ORGANIZATION_BLOCK "OB_TEST_AUTO"
TITLE = "Test Main — Simulacion Automatica TGBT V1.0"
{ S7_Optimized_Access := 'TRUE' }
// ============================================================================
// OB_TEST_AUTO  Ver 1.0  2026-03-13
//
// PROPÓSITO:
//   Validar la secuencia automática RED ↔ GD sin hardware real.
//   Reemplaza a OB1 (Main) durante la fase de prueba en taller/laboratorio.
//
// CÓMO ACTIVARLO EN TIA PORTAL (S7-1200):
//   1. Crear este bloque como "Organization Block → Program cycle" con un
//      número diferente a OB1 (ej: OB123).
//   2. En las propiedades de OB1 (Main), marcar "Unlinked" o agregar una
//      condición de retorno inmediato al inicio del bloque (IF NOT TEST_MODE THEN RETURN)
//      para que sólo corra uno de los dos ciclos.
//   3. Alternativamente: renombrar el "Main" actual y asignar este bloque
//      como el nuevo ciclo principal (número de OB = 1).
//
//   IMPORTANTE: NO ejecutar ambos OBs simultáneamente — ambos escriben
//   sobre las mismas instancias (02_FB_SCMTA_DB, 04_FB_CMD_ARBITER_DB, etc.)
//   lo que generaría resultados imprevisibles.
//
// QUÉ HACE ESTE OB vs OB1 (Main):
//   ✓ Llama a TEST_AUTO_FB en lugar de IO_NORMALIZE + Modbus Manager.
//     TEST_AUTO_FB inyecta directamente en DATA_BUFF:
//       - Mediciones de red simuladas (380V/50Hz ↔ 0V/0Hz)
//       - Señales GD1/GD2 (READY/RUNNING) como respuesta a %Q1.0/%Q1.1
//       - Feedback de interruptores como respuesta a pulsos %Q0.x
//   ✓ Llama a SCMTA con timers acortados:
//       T_MIN_GD_STAY  = 60 s   (producción: 10 min)
//       T_GRID_STABLE  = 30 s   (producción: 120 s)
//       T_GD_COOLDOWN  = 10 s   (producción: 60 s)
//   ✓ Llama a SHED, CMD_ARBITER, PULSE_EXPANDER, OUTPUTS igual que OB1.
//   ✗ NO llama a Modbus Manager (sin PM5350P).
//   ✗ NO llama a IO_NORMALIZE (TEST_AUTO_FB reemplaza esa función).
//
// CICLO DE PRUEBA AUTOMÁTICO (configurable en TEST_AUTO_DB):
//   T_FASE_GRID_OK  (30s) → RED OK  → SCMTA = ST_NORMAL_ON_GRID
//   Fin del timer          → RED FALLA (0V) → SCMTA inicia transferencia a GD
//   T_BRK_CONFIRM  (0.6s) → QT1 confirma apertura
//   Abre Q22               → T_BRK_CONFIRM → Q22 confirma apertura
//   T_START_GD_DELAY(3s)   → Arranque GD1 (%Q1.0←TRUE)
//   T_GD1_STARTUP  (8s)   → GD1_READY=TRUE, GD1_RUNNING=TRUE
//   T_GD_STABILIZATION(5s)→ SCMTA cierra QG1
//   T_BRK_CONFIRM  (0.6s) → QG1 confirma cierre → ST_ON_GD1
//   T_MIN_GD_STAY (60s)   → Espera mínima en GD antes de retorno
//   T_FASE_GRID_FAIL(90s) → Red se restaura (380V/50Hz)
//   T_GRID_STABLE  (30s)  → SCMTA abre QG1, cierra Q22, cierra QT1 → ST_ON_GRID
//   Ciclo se repite.
//
// CONTROLES HMI DURANTE PRUEBA (escribir en TEST_AUTO_DB):
//   TEST_AUTO_DB.FORCE_GRID_FAIL  := TRUE  → falla de red inmediata
//   TEST_AUTO_DB.FORCE_GRID_OK    := TRUE  → red restaurada inmediata
//   TEST_AUTO_DB.FORCE_GD1_ALARM  := TRUE  → alarma GD1 en marcha
//   DATA_BUFF.RESET_FAULT         := TRUE  → reset falla SCMTA
// ============================================================================
VERSION : 0.1

BEGIN

    // ========================================================================
    // NETWORK 1: IO REAL (CPU + EXPANSION)
    // Igual que OB1, pero forzando MODE_AUTO para prueba automática.
    // ========================================================================
    "01_FB_IO_NORMALIZE_DB"(
        DI_SYS_AUTO       := TRUE,

        // QT1 (CPU)
        DI_QT1_REMOTE     := %I0.0,
        DI_QT1_CLOSE      := %I0.1,
        DI_QT1_FAULT      := %I0.2,
        DI_QT1_UV_OV      := %I0.3,

        DI_BUSBAR_UV_OV   := %I0.4,

        // QG1 (CPU)
        DI_QG1_REMOTE     := %I0.5,
        DI_QG1_CLOSE      := %I0.6,
        DI_QG1_FAULT      := %I0.7,
        DI_QG1_UV_OV      := %I1.0,

        // QG2 (CPU)
        DI_QG2_REMOTE     := %I1.1,
        DI_QG2_CLOSE      := %I1.2,
        DI_QG2_FAULT      := %I1.3,
        DI_QG2_UV_OV      := %I1.4,

        // Q22 remoto (CPU)
        DI_Q22_REMOTE     := %I1.5,

        MODE_AUTO         => "DATA_BUFF".MODE_AUTO,
        MODE_MANUAL       => "DATA_BUFF".MODE_MANUAL,
        DIAG_MODE_VALID   => "DATA_BUFF".DIAG_MODE_VALID,

        QT1_CLOSED        => "DATA_BUFF".QT1_CLOSED,
        QT1_OPEN          => "DATA_BUFF".QT1_OPEN,
        QT1_FAULT         => "DATA_BUFF".QT1_FAULT,
        QT1_REMOTE        => "DATA_BUFF".QT1_REMOTE,
        QT1_UV_OV_DI      => "DATA_BUFF".QT1_UV_OV_DI,

        BUSBAR_UV_OV_DI   => "DATA_BUFF".BUSBAR_UV_OV_DI,

        QG1_CLOSED        => "DATA_BUFF".QG1_CLOSED,
        QG1_OPEN          => "DATA_BUFF".QG1_OPEN,
        QG1_FAULT         => "DATA_BUFF".QG1_FAULT,
        QG1_REMOTE        => "DATA_BUFF".QG1_REMOTE,
        QG1_UV_OV_DI      => "DATA_BUFF".QG1_UV_OV_DI,

        QG2_CLOSED        => "DATA_BUFF".QG2_CLOSED,
        QG2_OPEN          => "DATA_BUFF".QG2_OPEN,
        QG2_FAULT         => "DATA_BUFF".QG2_FAULT,
        QG2_REMOTE        => "DATA_BUFF".QG2_REMOTE,
        QG2_UV_OV_DI      => "DATA_BUFF".QG2_UV_OV_DI,

        Q22_REMOTE        => "DATA_BUFF".Q22_REMOTE
    );

    // En prueba usar la condición REMOTO real de DI, sin forzado.
    "DATA_BUFF".QT1_REMOTE_ALLOWED := "DATA_BUFF".QT1_REMOTE;
    "DATA_BUFF".QG1_REMOTE_ALLOWED := "DATA_BUFF".QG1_REMOTE;
    "DATA_BUFF".QG2_REMOTE_ALLOWED := "DATA_BUFF".QG2_REMOTE;
    "DATA_BUFF".Q22_REMOTE_ALLOWED := "DATA_BUFF".Q22_REMOTE;
    "DATA_BUFF".Q22_CLOSED := %I8.0;
    "DATA_BUFF".Q22_FAULT  := %I8.1;


    // ========================================================================
    // NETWORK 2: SIMULADOR DE RED/GD
    // Mantiene test automático de transferencia sin depender de Modbus real.
    // ========================================================================
    // Usar parámetros guardados en TEST_AUTO_DB para permitir ajuste online
    // (FORCE_GRID_FAIL, FORCE_GRID_OK, FORCE_GDx_ALARM, tiempos, etc.).
    "TEST_AUTO_DB"();


    // ========================================================================
    // NETWORK 3: MÁQUINA DE ESTADOS SCMTA
    // Misma instancia que OB1 → misma lógica de transferencia.
    // Timers reducidos para hacer el ciclo de prueba razonablemente rápido.
    // ========================================================================
    "02_FB_SCMTA_DB"(
        ENABLE               := TRUE,
        MODE_AUTO            := "DATA_BUFF".MODE_AUTO,
        ENABLE_QG2           := "DB_PARAMS".ENABLE_QG2,
        ENABLE_AUTO_RETURN   := TRUE,
        RESET_FAULT          := "DATA_BUFF".RESET_FAULT,

        // Posición/estado interruptores (provistos por TEST_AUTO_FB)
        QT1_CLOSED           := "DATA_BUFF".QT1_CLOSED,
        QT1_FAULT            := "DATA_BUFF".QT1_FAULT,
        QT1_REMOTE           := "DATA_BUFF".QT1_REMOTE,
        QT1_UV_OV_DI         := "DATA_BUFF".QT1_UV_OV_DI,

        QG1_CLOSED           := "DATA_BUFF".QG1_CLOSED,
        QG1_FAULT            := "DATA_BUFF".QG1_FAULT,
        QG1_REMOTE           := "DATA_BUFF".QG1_REMOTE,

        QG2_CLOSED           := "DATA_BUFF".QG2_CLOSED,
        QG2_FAULT            := "DATA_BUFF".QG2_FAULT,
        QG2_REMOTE           := "DATA_BUFF".QG2_REMOTE,

        Q22_CLOSED           := "DATA_BUFF".Q22_CLOSED,

        // Mediciones RED (provistos por TEST_AUTO_FB — sin Modbus)
        GRID_V_L1L2          := "DATA_BUFF".GRID_V_L1L2,
        GRID_V_L2L3          := "DATA_BUFF".GRID_V_L2L3,
        GRID_V_L3L1          := "DATA_BUFF".GRID_V_L3L1,
        GRID_FREQ            := "DATA_BUFF".GRID_FREQ,
        GRID_MEASUREMENT_OK  := "DATA_BUFF".GRID_MEASUREMENT_OK,
        GRID_PHASE_LOSS      := "DATA_BUFF".GRID_PHASE_LOSS,
        GRID_ALM_UV          := "DATA_BUFF".GRID_ALM_UV,
        GRID_ALM_OV          := "DATA_BUFF".GRID_ALM_OV,

        // Criterio GD por medicion electrica + Modbus OK (simulado por TEST_AUTO_FB)
        GD1_V_L1L2           := "DATA_BUFF".GD1_V_L1L2,
        GD1_V_L2L3           := "DATA_BUFF".GD1_V_L2L3,
        GD1_V_L3L1           := "DATA_BUFF".GD1_V_L3L1,
        GD1_FREQ             := "DATA_BUFF".GD1_FREQ,
        GD1_MEASUREMENT_OK   := "DATA_BUFF".GD1_MEASUREMENT_OK,
        GD2_V_L1L2           := "DATA_BUFF".GD2_V_L1L2,
        GD2_V_L2L3           := "DATA_BUFF".GD2_V_L2L3,
        GD2_V_L3L1           := "DATA_BUFF".GD2_V_L3L1,
        GD2_FREQ             := "DATA_BUFF".GD2_FREQ,
        GD2_MEASUREMENT_OK   := "DATA_BUFF".GD2_MEASUREMENT_OK,

        // Parámetros nominales de red (valores reales)
        V_NOM                := 380.0,
        V_MIN_PCT            := 85.0,
        V_MAX_PCT            := 110.0,
        FREQ_NOM             := 50.0,
        FREQ_MIN             := 49.0,
        FREQ_MAX             := 51.0,

        // Timers de transferencia RED→GD (valores reales de producción)
        T_OPEN_QT1           := T#3s,
        T_OPEN_Q22           := T#3s,
        T_DELAY_CLOSE_Q22    := T#10s,
        T_CLOSE_Q22          := T#3s,
        T_START_GD_DELAY     := T#3s,
        T_GD_READY_TIMEOUT   := T#30s,
        MAX_GD_START_RETRIES := 2,
        T_GD_STABILIZATION   := T#30s,
        T_CLOSE_QG1          := T#3s,
        T_CLOSE_QG2          := T#3s,
        T_CMD_CONFIRM        := T#2s,
        T_GRID_FAIL_FILTER   := T#2s,

        // Timers de retorno GD→RED  *** ACORTADOS PARA TEST ***
        // (en producción usar DB_PARAMS: T_MIN_GD_STAY=10min, T_GRID_STABLE=120s)
        T_MIN_GD_STAY        := T#10s,   // Test rápido de secuencia
        T_GRID_STABLE        := T#5s,    // Test rápido de retorno
        T_OPEN_QG1           := T#3s,
        T_OPEN_QG2           := T#3s,
        T_CLOSE_QT1          := T#3s,
        T_GD_COOLDOWN        := T#2s,    // Test rápido

        // Outputs → DATA_BUFF
        STATE                => "DATA_BUFF".SCMTA_STATE,
        STATE_NAME           => "DATA_BUFF".SCMTA_STATE_NAME,
        REQ_SCMTA_OPEN_QT1   => "02_FB_SCMTA_DB".REQ_SCMTA_OPEN_QT1,
        REQ_SCMTA_CLOSE_QT1  => "02_FB_SCMTA_DB".REQ_SCMTA_CLOSE_QT1,
        REQ_SCMTA_OPEN_QG1   => "02_FB_SCMTA_DB".REQ_SCMTA_OPEN_QG1,
        REQ_SCMTA_CLOSE_QG1  => "02_FB_SCMTA_DB".REQ_SCMTA_CLOSE_QG1,
        REQ_SCMTA_OPEN_QG2   => "02_FB_SCMTA_DB".REQ_SCMTA_OPEN_QG2,
        REQ_SCMTA_CLOSE_QG2  => "02_FB_SCMTA_DB".REQ_SCMTA_CLOSE_QG2,
        REQ_SCMTA_OPEN_Q22   => "02_FB_SCMTA_DB".REQ_SCMTA_OPEN_Q22,
        REQ_SCMTA_CLOSE_Q22  => "02_FB_SCMTA_DB".REQ_SCMTA_CLOSE_Q22,
        DO_GD_START          => %Q1.0,
        DO_GD_STOP           => "DATA_BUFF".GD_STOP_REQ,
        DO_GD2_START         => %Q1.1,
        DO_GD2_STOP          => "DATA_BUFF".GD2_STOP_REQ,
        IS_ON_GRID           => "DATA_BUFF".IS_ON_GRID,
        IS_ON_GD             => "DATA_BUFF".IS_ON_GD,
        IS_ON_GD1            => "DATA_BUFF".IS_ON_GD1,
        IS_ON_GD2            => "DATA_BUFF".IS_ON_GD2,
        ACTIVE_GD            => "DATA_BUFF".ACTIVE_GD,
        IS_IN_TRANSFER       => "DATA_BUFF".IS_IN_TRANSFER,
        IS_FAULT             => "DATA_BUFF".IS_FAULT,
        TRANSFER_TO_GD       => "DATA_BUFF".TRANSFER_TO_GD,
        GRID_OK              => "DATA_BUFF".GRID_OK,
        GRID_FAIL            => "DATA_BUFF".GRID_FAIL,
        FAULT_CODE           => "DATA_BUFF".FAULT_CODE,
        ELAPSED_TIME         => "DATA_BUFF".ELAPSED_TIME,
        DIAG_LAST_TRANSFER_TIME => "DATA_BUFF".DIAG_LAST_TRANSFER_TIME,
        GD1_AVAILABLE        => "DATA_BUFF".GD1_AVAILABLE,
        GD2_AVAILABLE        => "DATA_BUFF".GD2_AVAILABLE
    );

    // GD STOP: limpiar %Q1.x cuando SCMTA solicita parada
    IF "DATA_BUFF".GD_STOP_REQ  THEN %Q1.0 := FALSE; END_IF;
    IF "DATA_BUFF".GD2_STOP_REQ THEN %Q1.1 := FALSE; END_IF;


    // ========================================================================
    // NETWORK 4: DESLASTRE (deshabilitado en prueba)
    // ========================================================================
    "03_FB_SHED_DB"(
        ENABLE              := FALSE,
        MODE_AUTO           := "DATA_BUFF".MODE_AUTO,
        IS_ON_GD            := "DATA_BUFF".IS_ON_GD,
        IS_ON_GRID          := "DATA_BUFF".IS_ON_GRID,
        IS_IN_TRANSFER      := "DATA_BUFF".IS_IN_TRANSFER,
        TRANSFER_TO_GD      := "DATA_BUFF".TRANSFER_TO_GD,
        GD_LoadPct          := 0.0,
        TR_LoadPct          := 0.0,
        GD_SHED_ON          := "DB_PARAMS".GD_SHED_ON,
        GD_SHED_OFF         := "DB_PARAMS".GD_SHED_OFF,
        GRID_SHED_ON        := "DB_PARAMS".GRID_SHED_ON,
        GRID_SHED_OFF       := "DB_PARAMS".GRID_SHED_OFF,
        T_SHED_STEP         := "DB_PARAMS".T_SHED_STEP,
        T_RECONNECT_STEP    := "DB_PARAMS".T_RECONNECT_STEP,
        T_LOAD_FILTER       := "DB_PARAMS".T_LOAD_FILTER,
        T_LOAD_CHECK_DELAY  := "DB_PARAMS".T_LOAD_CHECK_DELAY,
        SHED_ORDER          := "DB_PARAMS".SHED_ORDER,
        RECONNECT_ORDER     := "DB_PARAMS".RECONNECT_ORDER,
        FEEDER_ESSENTIAL    := "DB_PARAMS".FEEDER_ESSENTIAL,
        SHED_ENABLE         := "DB_PARAMS".SHED_ENABLE,
        FEEDER_STATE        := "DB_PARAMS".SHED_ORDER,
        SHED_ACTIVE         => "DATA_BUFF".SHED_ACTIVE
    );


    // ========================================================================
    // NETWORK 5: ÁRBITRO DE COMANDOS
    // ========================================================================
    "04_FB_CMD_ARBITER_DB"(
        REQ_SCMTA_OPEN_QT1  := "02_FB_SCMTA_DB".REQ_SCMTA_OPEN_QT1,
        REQ_SCMTA_CLOSE_QT1 := "02_FB_SCMTA_DB".REQ_SCMTA_CLOSE_QT1,
        REQ_SCMTA_OPEN_QG1  := "02_FB_SCMTA_DB".REQ_SCMTA_OPEN_QG1,
        REQ_SCMTA_CLOSE_QG1 := "02_FB_SCMTA_DB".REQ_SCMTA_CLOSE_QG1,
        REQ_SCMTA_OPEN_QG2  := "02_FB_SCMTA_DB".REQ_SCMTA_OPEN_QG2,
        REQ_SCMTA_CLOSE_QG2 := "02_FB_SCMTA_DB".REQ_SCMTA_CLOSE_QG2,
        REQ_SCMTA_OPEN_Q22  := "02_FB_SCMTA_DB".REQ_SCMTA_OPEN_Q22,
        REQ_SCMTA_CLOSE_Q22 := "02_FB_SCMTA_DB".REQ_SCMTA_CLOSE_Q22,
        REQ_MAN_QT1_OPEN    := "DATA_BUFF".REQ_MAN_QT1_OPEN,
        REQ_MAN_QT1_CLOSE   := "DATA_BUFF".REQ_MAN_QT1_CLOSE,
        REQ_MAN_QG1_OPEN    := "DATA_BUFF".REQ_MAN_QG1_OPEN,
        REQ_MAN_QG1_CLOSE   := "DATA_BUFF".REQ_MAN_QG1_CLOSE,
        REQ_MAN_QG2_OPEN    := "DATA_BUFF".REQ_MAN_QG2_OPEN,
        REQ_MAN_QG2_CLOSE   := "DATA_BUFF".REQ_MAN_QG2_CLOSE,
        REQ_MAN_Q22_OPEN    := "DATA_BUFF".REQ_MAN_Q22_OPEN,
        REQ_MAN_Q22_CLOSE   := "DATA_BUFF".REQ_MAN_Q22_CLOSE,
        MODE_AUTO           := "DATA_BUFF".MODE_AUTO,
        MODE_MANUAL         := "DATA_BUFF".MODE_MANUAL,
        QT1_CLOSED          := "DATA_BUFF".QT1_CLOSED,
        QG1_CLOSED          := "DATA_BUFF".QG1_CLOSED,
        QG2_CLOSED          := "DATA_BUFF".QG2_CLOSED,
        QT1_REMOTE          := "DATA_BUFF".QT1_REMOTE_ALLOWED,
        QG1_REMOTE          := "DATA_BUFF".QG1_REMOTE_ALLOWED,
        QG2_REMOTE          := "DATA_BUFF".QG2_REMOTE_ALLOWED,
        Q22_REMOTE          := "DATA_BUFF".Q22_REMOTE_ALLOWED,
        BLOCK_LOCAL         => "DATA_BUFF".BLOCK_LOCAL,
        BLOCK_INTERLOCK     => "DATA_BUFF".BLOCK_INTERLOCK,
        BLOCK_CONFLICT      => "DATA_BUFF".BLOCK_CONFLICT,
        ALM_INTERLOCK_VIOLATION := "DATA_BUFF".ALM_INTERLOCK_VIOLATION
    );


    // ========================================================================
    // NETWORK 6: PULSE EXPANDER — CMD (1 scan) → DO pulso 300 ms
    // %Q0.0=CLOSE_QT1  %Q0.1=OPEN_QT1
    // %Q0.2=CLOSE_QG1  %Q0.3=OPEN_QG1
    // %Q0.4=CLOSE_QG2  %Q0.5=OPEN_QG2
    // %Q0.6=CLOSE_Q22  %Q0.7=OPEN_Q22
    // ========================================================================
    "12_PULSE_EXPANDER_DB"(
        T_PULSE  := T#300ms,
        TRIG_1   := "04_FB_CMD_ARBITER_DB".CMD_CLOSE_QT1,
        TRIG_2   := "04_FB_CMD_ARBITER_DB".CMD_OPEN_QT1,
        TRIG_3   := "04_FB_CMD_ARBITER_DB".CMD_CLOSE_QG1,
        TRIG_4   := "04_FB_CMD_ARBITER_DB".CMD_OPEN_QG1,
        TRIG_5   := "04_FB_CMD_ARBITER_DB".CMD_CLOSE_QG2,
        TRIG_6   := "04_FB_CMD_ARBITER_DB".CMD_OPEN_QG2,
        TRIG_7   := "04_FB_CMD_ARBITER_DB".CMD_CLOSE_Q22,
        TRIG_8   := "04_FB_CMD_ARBITER_DB".CMD_OPEN_Q22,
        OUT_1    => %Q0.0,
        OUT_2    => %Q0.1,
        OUT_3    => %Q0.2,
        OUT_4    => %Q0.3,
        OUT_5    => %Q0.4,
        OUT_6    => %Q0.5,
        OUT_7    => %Q0.6,
        OUT_8    => %Q0.7
    );

    // Espejo a DQ de expansión para validar salidas en ambos bornes
    %Q8.0 := %Q0.0;
    %Q8.1 := %Q0.1;
    %Q8.2 := %Q0.2;
    %Q8.3 := %Q0.3;
    %Q8.4 := %Q0.4;
    %Q8.5 := %Q0.5;
    %Q8.6 := %Q0.6;
    %Q8.7 := %Q0.7;


    // ========================================================================
    // NETWORK 7: SALIDAS PILOTO / HMI  (05_FB_OUTPUTS)
    // ========================================================================
    "05_FB_OUTPUTS_DB"(
        IS_ON_GRID     := "DATA_BUFF".IS_ON_GRID,
        IS_ON_GD       := "DATA_BUFF".IS_ON_GD,
        IS_IN_TRANSFER := "DATA_BUFF".IS_IN_TRANSFER,
        IS_FAULT       := "DATA_BUFF".IS_FAULT,
        STATE          := "DATA_BUFF".SCMTA_STATE,
        STATE_NAME     := "DATA_BUFF".SCMTA_STATE_NAME,
        FAULT_CODE     := "DATA_BUFF".FAULT_CODE,
        QT1_CLOSED     := "DATA_BUFF".QT1_CLOSED,
        QT1_FAULT      := "DATA_BUFF".QT1_FAULT,
        QG1_CLOSED     := "DATA_BUFF".QG1_CLOSED,
        QG1_FAULT      := "DATA_BUFF".QG1_FAULT,
        QG2_CLOSED     := "DATA_BUFF".QG2_CLOSED,
        QG2_FAULT      := "DATA_BUFF".QG2_FAULT,
        Q22_CLOSED     := "DATA_BUFF".Q22_CLOSED,
        Q22_FAULT      := "DATA_BUFF".Q22_FAULT,
        ALM_INTERLOCK_VIOLATION := "DATA_BUFF".ALM_INTERLOCK_VIOLATION,
        BLOCK_INTERLOCK := "DATA_BUFF".BLOCK_INTERLOCK,
        GRID_FAIL      := "DATA_BUFF".GRID_FAIL,
        ACK_ALARM      := "DATA_BUFF".ACK_ALARM,
        DO_PILOT_ON_GRID    => "DATA_BUFF".PILOT_ON_GRID,
        DO_PILOT_ON_GD      => "DATA_BUFF".PILOT_ON_GD,
        DO_PILOT_FAULT      => "DATA_BUFF".PILOT_FAULT,
        DO_PILOT_QT1_OPEN   => "DATA_BUFF".PILOT_QT1_OPEN,
        DO_PILOT_QT1_CLOSED => "DATA_BUFF".PILOT_QT1_CLOSED,
        DO_PILOT_QT1_FAULT  => "DATA_BUFF".PILOT_QT1_FAULT,
        DO_PILOT_QG1_OPEN   => "DATA_BUFF".PILOT_QG1_OPEN,
        DO_PILOT_QG1_CLOSED => "DATA_BUFF".PILOT_QG1_CLOSED,
        DO_PILOT_QG1_FAULT  => "DATA_BUFF".PILOT_QG1_FAULT,
        DO_PILOT_QG2_OPEN   => "DATA_BUFF".PILOT_QG2_OPEN,
        DO_PILOT_QG2_CLOSED => "DATA_BUFF".PILOT_QG2_CLOSED,
        DO_PILOT_QG2_FAULT  => "DATA_BUFF".PILOT_QG2_FAULT,
        DO_PILOT_Q22_OPEN   => "DATA_BUFF".PILOT_Q22_OPEN,
        DO_PILOT_Q22_CLOSED => "DATA_BUFF".PILOT_Q22_CLOSED,
        DO_PILOT_Q22_FAULT  => "DATA_BUFF".PILOT_Q22_FAULT,
        DO_ALARM_BEACON     => %Q1.2,
        HMI_STATUS_TEXT     => "DATA_BUFF".SCMTA_STATE_NAME,
        HMI_ALARM_ACTIVE    => "DATA_BUFF".HMI_ALARM_ACTIVE,
        HMI_ALARM_TEXT      => "DATA_BUFF".HMI_ALARM_TEXT
    );

END_ORGANIZATION_BLOCK
